(* PLC project SafeLOGIC-1, BrAutomation SafeDESIGNER  4.2.0.17 *)
(* stored: companyURL http://www.br-automation.com, creationDateTime Tue Sep 13 10:12:13 2016 *)

PROGRAM Main

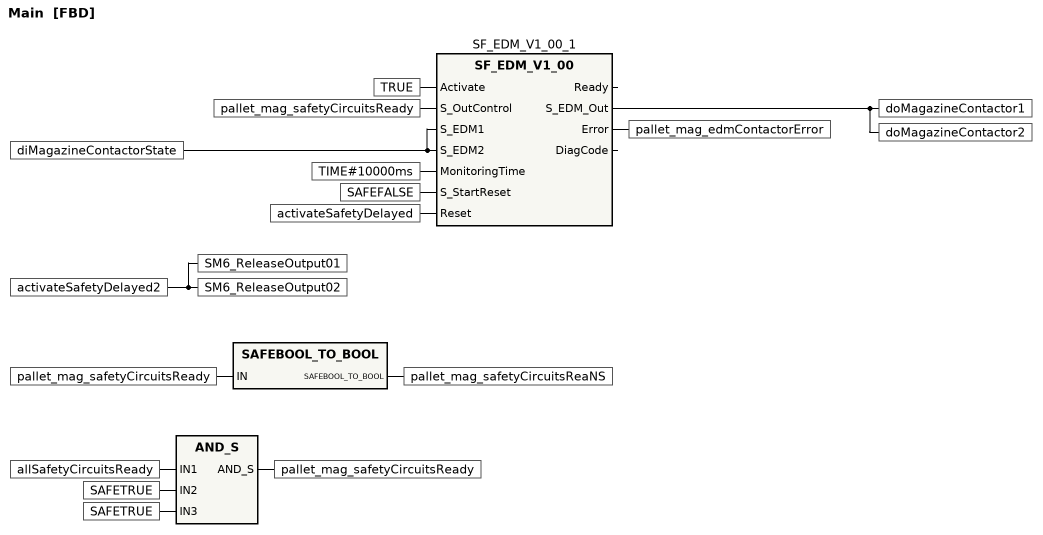
(* FBD diagram, written out as Structured Text *)
pallet_mag_safetyCircuitsReady := AND_S(allSafetyCircuitsReady, SAFETRUE, SAFETRUE);
SF_EDM_V1_00_1(Activate := TRUE, S_OutControl := pallet_mag_safetyCircuitsReady, S_EDM1 := diMagazineContactorState, S_EDM2 := diMagazineContactorState, MonitoringTime := TIME#10000ms, S_StartReset := SAFEFALSE, Reset := activateSafetyDelayed);
pallet_mag_edmContactorError := SF_EDM_V1_00_1.Error;
doMagazineContactor1 := SF_EDM_V1_00_1.S_EDM_Out;
doMagazineContactor2 := SF_EDM_V1_00_1.S_EDM_Out;
SM6_ReleaseOutput02 := activateSafetyDelayed2;
SM6_ReleaseOutput01 := activateSafetyDelayed2;
pallet_mag_safetyCircuitsReaNS := SAFEBOOL_TO_BOOL(pallet_mag_safetyCircuitsReady);
END_PROGRAM
